// TIA Portal V15 export
// export: Created 2018-12-10T18:36:37.9324983Z, ExportSetting WithDefaults, WithReadOnly, DisplayName Totally Integrated Automation Portal, DisplayVersion V15 Update 2, DisplayName TIA Portal Openness, DisplayVersion V15 Update 2, DisplayName STEP 7 Professional, DisplayVersion V15 Update 2, DisplayName STEP 7 Safety, DisplayVersion V15, DisplayName WinCC Professional, DisplayVersion V15 Update 2, DisplayName SIMATIC Visualization Architect, DisplayVersion V15 Update 1
DATA_BLOCK "FGDB_FIXTURENAME@AddOn"   // DB132
TITLE = Geostation addon-info / Geostation Zusatz-Info
{ S7_Optimized_Access := 'FALSE' }
AUTHOR : integra
FAMILY : SYS
VERSION : 0.51
// stored: AutoNumber true, CodeModifiedDate 2017-10-24T16:57:02.4799433Z, CompileDate 2018-02-20T10:24:36.1111751Z, CreationDate 2016-12-16T08:19:31.4249609Z, DBAccessibleFromOPCUA true, InterfaceModifiedDate 2017-10-24T16:57:02.4799433Z, IsConsistent true, IsKnowHowProtected false, IsOnlyStoredInLoadMemory false, IsPLCDB false, IsWriteProtectedInAS false, ModifiedDate 2018-01-29T16:41:32.7806867Z, ParameterModified 2017-10-24T16:57:02.4799433Z, StructureModified 2017-10-24T16:57:02.4799433Z
   VAR RETAIN
      AddInfo { ExternalAccessible := 'False'; ExternalVisible := 'False'; ExternalWritable := 'False'} : Struct   // Additional informations / Zusätzliche Informationen
         "1" { ExternalAccessible := 'False'; ExternalVisible := 'False'; ExternalWritable := 'False'} : DWord;   // Additional information 1 / Zusätzliche Information 1
         "2" { ExternalAccessible := 'False'; ExternalVisible := 'False'; ExternalWritable := 'False'} : DWord;   // Additional information 2 / Zusätzliche Information 2
         "3" { ExternalAccessible := 'False'; ExternalVisible := 'False'; ExternalWritable := 'False'} : DWord;   // Additional information 3 / Zusätzliche Information 3
         "4" { ExternalAccessible := 'False'; ExternalVisible := 'False'; ExternalWritable := 'False'} : DWord;   // Additional information 4 / Zusätzliche Information 4
         "5" { ExternalAccessible := 'False'; ExternalVisible := 'False'; ExternalWritable := 'False'} : DWord;   // Additional information 5 / Zusätzliche Information 5
         "6" { ExternalAccessible := 'False'; ExternalVisible := 'False'; ExternalWritable := 'False'} : DWord;   // Additional information 6 / Zusätzliche Information 6
      END_STRUCT;
      AddT { ExternalAccessible := 'False'; ExternalVisible := 'False'; ExternalWritable := 'False'} : Struct   // Additional tags / Zusätzliche Steuervariablen
         "1" { ExternalAccessible := 'False'; ExternalVisible := 'False'; ExternalWritable := 'False'} : Bool;   // !* Additional tag 1 / !* Zusätzliche Steuervariablen 1
         "2" { ExternalAccessible := 'False'; ExternalVisible := 'False'; ExternalWritable := 'False'} : Bool;   // !* Additional tag 2 / !* Zusätzliche Steuervariablen 2
         "3" { ExternalAccessible := 'False'; ExternalVisible := 'False'; ExternalWritable := 'False'} : Bool;   // !* Additional tag 3 / !* Zusätzliche Steuervariablen 3
         "4" { ExternalAccessible := 'False'; ExternalVisible := 'False'; ExternalWritable := 'False'} : Bool;   // !* Additional tag 4 / !* Zusätzliche Steuervariablen 4
         "5" { ExternalAccessible := 'False'; ExternalVisible := 'False'; ExternalWritable := 'False'} : Bool;   // !* Additional tag 5 / !* Zusätzliche Steuervariablen 5
         "6" { ExternalAccessible := 'False'; ExternalVisible := 'False'; ExternalWritable := 'False'} : Bool;   // !* Additional tag 6 / !* Zusätzliche Steuervariablen 6
         "7" { ExternalAccessible := 'False'; ExternalVisible := 'False'; ExternalWritable := 'False'} : Bool;   // !* Additional tag 7 / !* Zusätzliche Steuervariablen 7
         "8" { ExternalAccessible := 'False'; ExternalVisible := 'False'; ExternalWritable := 'False'} : Bool;   // !* Additional tag 8 / !* Zusätzliche Steuervariablen 8
         "9" { ExternalAccessible := 'False'; ExternalVisible := 'False'; ExternalWritable := 'False'} : Bool;   // !* Additional tag 9 / !* Zusätzliche Steuervariablen 9
         "10" { ExternalAccessible := 'False'; ExternalVisible := 'False'; ExternalWritable := 'False'} : Bool;   // !* Additional tag 10 / !* Zusätzliche Steuervariablen 10
         "11" { ExternalAccessible := 'False'; ExternalVisible := 'False'; ExternalWritable := 'False'} : Bool;   // !* Additional tag 11 / !* Zusätzliche Steuervariablen 11
         "12" { ExternalAccessible := 'False'; ExternalVisible := 'False'; ExternalWritable := 'False'} : Bool;   // !* Additional tag 12 / !* Zusätzliche Steuervariablen 12
         "13" { ExternalAccessible := 'False'; ExternalVisible := 'False'; ExternalWritable := 'False'} : Bool;   // !* Additional tag 13 / !* Zusätzliche Steuervariablen 13
         "14" { ExternalAccessible := 'False'; ExternalVisible := 'False'; ExternalWritable := 'False'} : Bool;   // !* Additional tag 14 / !* Zusätzliche Steuervariablen 14
         "15" { ExternalAccessible := 'False'; ExternalVisible := 'False'; ExternalWritable := 'False'} : Bool;   // !* Additional tag 15 / !* Zusätzliche Steuervariablen 15
         "16" { ExternalAccessible := 'False'; ExternalVisible := 'False'; ExternalWritable := 'False'} : Bool;   // !* Additional tag 16 / !* Zusätzliche Steuervariablen 16
      END_STRUCT;
      AddS { ExternalAccessible := 'False'; ExternalVisible := 'False'; ExternalWritable := 'False'} : Struct   // Additional sensors / Zusätzliche Sensoren
         init_pos { ExternalAccessible := 'False'; ExternalVisible := 'False'; ExternalWritable := 'False'} : Bool;   // initial position station empty / Anfangsposition Station leer
         "2" { ExternalAccessible := 'False'; ExternalVisible := 'False'; ExternalWritable := 'False'} : Bool;   // !* Additional tag 2 / !* Zusätzliche Steuervariablen 2
         "3" { ExternalAccessible := 'False'; ExternalVisible := 'False'; ExternalWritable := 'False'} : Bool;   // !* Additional tag 3 / !* Zusätzliche Steuervariablen 3
         "4" { ExternalAccessible := 'False'; ExternalVisible := 'False'; ExternalWritable := 'False'} : Bool;   // !* Additional tag 4 / !* Zusätzliche Steuervariablen 4
         "5" { ExternalAccessible := 'False'; ExternalVisible := 'False'; ExternalWritable := 'False'} : Bool;   // !* Additional tag 5 / !* Zusätzliche Steuervariablen 5
         "6" { ExternalAccessible := 'False'; ExternalVisible := 'False'; ExternalWritable := 'False'} : Bool;   // !* Additional tag 6 / !* Zusätzliche Steuervariablen 6
         "7" { ExternalAccessible := 'False'; ExternalVisible := 'False'; ExternalWritable := 'False'} : Bool;   // !* Additional tag 7 / !* Zusätzliche Steuervariablen 7
         "8" { ExternalAccessible := 'False'; ExternalVisible := 'False'; ExternalWritable := 'False'} : Bool;   // !* Additional tag 8 / !* Zusätzliche Steuervariablen 8
         "9" { ExternalAccessible := 'False'; ExternalVisible := 'False'; ExternalWritable := 'False'} : Bool;   // !* Additional tag 9 / !* Zusätzliche Steuervariablen 9
         "10" { ExternalAccessible := 'False'; ExternalVisible := 'False'; ExternalWritable := 'False'} : Bool;   // !* Additional tag 10 / !* Zusätzliche Steuervariablen 10
         "11" { ExternalAccessible := 'False'; ExternalVisible := 'False'; ExternalWritable := 'False'} : Bool;   // !* Additional tag 11 / !* Zusätzliche Steuervariablen 11
         "12" { ExternalAccessible := 'False'; ExternalVisible := 'False'; ExternalWritable := 'False'} : Bool;   // !* Additional tag 12 / !* Zusätzliche Steuervariablen 12
         "13" { ExternalAccessible := 'False'; ExternalVisible := 'False'; ExternalWritable := 'False'} : Bool;   // !* Additional tag 13 / !* Zusätzliche Steuervariablen 13
         "14" { ExternalAccessible := 'False'; ExternalVisible := 'False'; ExternalWritable := 'False'} : Bool;   // !* Additional tag 14 / !* Zusätzliche Steuervariablen 14
         "15" { ExternalAccessible := 'False'; ExternalVisible := 'False'; ExternalWritable := 'False'} : Bool;   // !* Additional tag 15 / !* Zusätzliche Steuervariablen 15
         "16" { ExternalAccessible := 'False'; ExternalVisible := 'False'; ExternalWritable := 'False'} : Bool;   // !* Additional tag 16 / !* Zusätzliche Steuervariablen 16
      END_STRUCT;
      ExtF { ExternalAccessible := 'False'; ExternalVisible := 'False'; ExternalWritable := 'False'} : Struct   // External faults / Externe Störungen
         PartControl { ExternalAccessible := 'False'; ExternalVisible := 'False'; ExternalWritable := 'False'} : Bool;   // Part Control Error / Bauteilkontrol Fehler
         "2" { ExternalAccessible := 'False'; ExternalVisible := 'False'; ExternalWritable := 'False'} : Bool;   // !* External fault 2 / !* Externer Störung 2
         "3" { ExternalAccessible := 'False'; ExternalVisible := 'False'; ExternalWritable := 'False'} : Bool;   // !* External fault 3 / !* Externer Störung 3
         "4" { ExternalAccessible := 'False'; ExternalVisible := 'False'; ExternalWritable := 'False'} : Bool;   // !* External fault 4 / !* Externer Störung 4
         "5" { ExternalAccessible := 'False'; ExternalVisible := 'False'; ExternalWritable := 'False'} : Bool;   // !* External fault 5 / !* Externer Störung 5
         "6" { ExternalAccessible := 'False'; ExternalVisible := 'False'; ExternalWritable := 'False'} : Bool;   // !* External fault 6 / !* Externer Störung 6
         "7" { ExternalAccessible := 'False'; ExternalVisible := 'False'; ExternalWritable := 'False'} : Bool;   // !* External fault 7 / !* Externer Störung 7
         "8" { ExternalAccessible := 'False'; ExternalVisible := 'False'; ExternalWritable := 'False'} : Bool;   // !* External fault 8 / !* Externer Störung 8
         "9" { ExternalAccessible := 'False'; ExternalVisible := 'False'; ExternalWritable := 'False'} : Bool;   // !* External fault 9 / !* Externer Störung 9
         "10" { ExternalAccessible := 'False'; ExternalVisible := 'False'; ExternalWritable := 'False'} : Bool;   // !* External fault 10 / !* Externer Störung 10
         "11" { ExternalAccessible := 'False'; ExternalVisible := 'False'; ExternalWritable := 'False'} : Bool;   // !* External fault 11 / !* Externer Störung 11
         "12" { ExternalAccessible := 'False'; ExternalVisible := 'False'; ExternalWritable := 'False'} : Bool;   // !* External fault 12 / !* Externer Störung 12
         "13" { ExternalAccessible := 'False'; ExternalVisible := 'False'; ExternalWritable := 'False'} : Bool;   // !* External fault 13 / !* Externer Störung 13
         "14" { ExternalAccessible := 'False'; ExternalVisible := 'False'; ExternalWritable := 'False'} : Bool;   // !* External fault 14 / !* Externer Störung 14
         "15" { ExternalAccessible := 'False'; ExternalVisible := 'False'; ExternalWritable := 'False'} : Bool;   // !* External fault 15 / !* Externer Störung 15
         "16" { ExternalAccessible := 'False'; ExternalVisible := 'False'; ExternalWritable := 'False'} : Bool;   // !* External fault 16 / !* Externer Störung 16
      END_STRUCT;
      TransExtF { ExternalAccessible := 'False'; ExternalVisible := 'False'; ExternalWritable := 'False'} : Struct   // Transfer external faults / Übergabe externe Störungen
         PartControl { ExternalAccessible := 'False'; ExternalVisible := 'False'; ExternalWritable := 'False'} : Bool;   // Transfer external fault PartControl / Übergabe externer Störung Bauteilkontrol
         "2" { ExternalAccessible := 'False'; ExternalVisible := 'False'; ExternalWritable := 'False'} : Bool;   // Transfer external fault 2 / Übergabe externer Störung 2
         "3" { ExternalAccessible := 'False'; ExternalVisible := 'False'; ExternalWritable := 'False'} : Bool;   // Transfer external fault 3 / Übergabe externer Störung 3
         "4" { ExternalAccessible := 'False'; ExternalVisible := 'False'; ExternalWritable := 'False'} : Bool;   // Transfer external fault 4 / Übergabe externer Störung 4
         "5" { ExternalAccessible := 'False'; ExternalVisible := 'False'; ExternalWritable := 'False'} : Bool;   // Transfer external fault 5 / Übergabe externer Störung 5
         "6" { ExternalAccessible := 'False'; ExternalVisible := 'False'; ExternalWritable := 'False'} : Bool;   // Transfer external fault 6 / Übergabe externer Störung 6
         "7" { ExternalAccessible := 'False'; ExternalVisible := 'False'; ExternalWritable := 'False'} : Bool;   // Transfer external fault 7 / Übergabe externer Störung 7
         "8" { ExternalAccessible := 'False'; ExternalVisible := 'False'; ExternalWritable := 'False'} : Bool;   // Transfer external fault 8 / Übergabe externer Störung 8
         "9" { ExternalAccessible := 'False'; ExternalVisible := 'False'; ExternalWritable := 'False'} : Bool;   // Transfer external fault 9 / Übergabe externer Störung 9
         "10" { ExternalAccessible := 'False'; ExternalVisible := 'False'; ExternalWritable := 'False'} : Bool;   // Transfer external fault 10 / Übergabe externer Störung 10
         "11" { ExternalAccessible := 'False'; ExternalVisible := 'False'; ExternalWritable := 'False'} : Bool;   // Transfer external fault 11 / Übergabe externer Störung 11
         "12" { ExternalAccessible := 'False'; ExternalVisible := 'False'; ExternalWritable := 'False'} : Bool;   // Transfer external fault 12 / Übergabe externer Störung 12
         "13" { ExternalAccessible := 'False'; ExternalVisible := 'False'; ExternalWritable := 'False'} : Bool;   // Transfer external fault 13 / Übergabe externer Störung 13
         "14" { ExternalAccessible := 'False'; ExternalVisible := 'False'; ExternalWritable := 'False'} : Bool;   // Transfer external fault 14 / Übergabe externer Störung 14
         "15" { ExternalAccessible := 'False'; ExternalVisible := 'False'; ExternalWritable := 'False'} : Bool;   // Transfer external fault 15 / Übergabe externer Störung 15
         "16" { ExternalAccessible := 'False'; ExternalVisible := 'False'; ExternalWritable := 'False'} : Bool;   // Transfer external fault 16 / Übergabe externer Störung 16
      END_STRUCT;
      ExtW { ExternalAccessible := 'False'; ExternalVisible := 'False'; ExternalWritable := 'False'} : Struct   // External warnings / Externe Warnungen
         "1" { ExternalAccessible := 'False'; ExternalVisible := 'False'; ExternalWritable := 'False'} : Bool;   // !* External warning 1 / !* Externe Warnung 1
         "2" { ExternalAccessible := 'False'; ExternalVisible := 'False'; ExternalWritable := 'False'} : Bool;   // !* External warning 2 / !* Externe Warnung 2
         "3" { ExternalAccessible := 'False'; ExternalVisible := 'False'; ExternalWritable := 'False'} : Bool;   // !* External warning 3 / !* Externe Warnung 3
         "4" { ExternalAccessible := 'False'; ExternalVisible := 'False'; ExternalWritable := 'False'} : Bool;   // !* External warning 4 / !* Externe Warnung 4
         "5" { ExternalAccessible := 'False'; ExternalVisible := 'False'; ExternalWritable := 'False'} : Bool;   // !* External warning 5 / !* Externe Warnung 5
         "6" { ExternalAccessible := 'False'; ExternalVisible := 'False'; ExternalWritable := 'False'} : Bool;   // !* External warning 6 / !* Externe Warnung 6
         "7" { ExternalAccessible := 'False'; ExternalVisible := 'False'; ExternalWritable := 'False'} : Bool;   // !* External warning 7 / !* Externe Warnung 7
         "8" { ExternalAccessible := 'False'; ExternalVisible := 'False'; ExternalWritable := 'False'} : Bool;   // !* External warning 7 / !* Externe Warnung 7
      END_STRUCT;
      TransExtW { ExternalAccessible := 'False'; ExternalVisible := 'False'; ExternalWritable := 'False'} : Struct   // Transfer external warnings / Übergabe externe Warnungen
         "1" { ExternalAccessible := 'False'; ExternalVisible := 'False'; ExternalWritable := 'False'} : Bool;   // Transfer external warning 1 / Übergabe externe Warnung 1
         "2" { ExternalAccessible := 'False'; ExternalVisible := 'False'; ExternalWritable := 'False'} : Bool;   // Transfer external warning 2 / Übergabe externe Warnung 2
         "3" { ExternalAccessible := 'False'; ExternalVisible := 'False'; ExternalWritable := 'False'} : Bool;   // Transfer external warning 3 / Übergabe externe Warnung 3
         "4" { ExternalAccessible := 'False'; ExternalVisible := 'False'; ExternalWritable := 'False'} : Bool;   // Transfer external warning 4 / Übergabe externe Warnung 4
         "5" { ExternalAccessible := 'False'; ExternalVisible := 'False'; ExternalWritable := 'False'} : Bool;   // Transfer external warning 5 / Übergabe externe Warnung 5
         "6" { ExternalAccessible := 'False'; ExternalVisible := 'False'; ExternalWritable := 'False'} : Bool;   // Transfer external warning 6 / Übergabe externe Warnung 6
         "7" { ExternalAccessible := 'False'; ExternalVisible := 'False'; ExternalWritable := 'False'} : Bool;   // Transfer external warning 7 / Übergabe externe Warnung 7
         "8" { ExternalAccessible := 'False'; ExternalVisible := 'False'; ExternalWritable := 'False'} : Bool;   // Transfer external warning 8 / Übergabe externe Warnung 8
      END_STRUCT;
      ExtM { ExternalAccessible := 'False'; ExternalVisible := 'False'; ExternalWritable := 'False'} : Struct   // External messages / Externe Meldungen
         "1" { ExternalAccessible := 'False'; ExternalVisible := 'False'; ExternalWritable := 'False'} : Bool;   // !* External message 1 / !* Externe Meldung 1
         "2" { ExternalAccessible := 'False'; ExternalVisible := 'False'; ExternalWritable := 'False'} : Bool;   // !* External message 2 / !* Externe Meldung 2
         "3" { ExternalAccessible := 'False'; ExternalVisible := 'False'; ExternalWritable := 'False'} : Bool;   // !* External message 3 / !* Externe Meldung 3
         "4" { ExternalAccessible := 'False'; ExternalVisible := 'False'; ExternalWritable := 'False'} : Bool;   // !* External message 4 / !* Externe Meldung 4
         "5" { ExternalAccessible := 'False'; ExternalVisible := 'False'; ExternalWritable := 'False'} : Bool;   // !* External message 5 / !* Externe Meldung 5
         "6" { ExternalAccessible := 'False'; ExternalVisible := 'False'; ExternalWritable := 'False'} : Bool;   // !* External message 6 / !* Externe Meldung 6
         "7" { ExternalAccessible := 'False'; ExternalVisible := 'False'; ExternalWritable := 'False'} : Bool;   // !* External message 7 / !* Externe Meldung 7
         "8" { ExternalAccessible := 'False'; ExternalVisible := 'False'; ExternalWritable := 'False'} : Bool;   // !* External message 8 / !* Externe Meldung 8
      END_STRUCT;
      TransExtM { ExternalAccessible := 'False'; ExternalVisible := 'False'; ExternalWritable := 'False'} : Struct   // Transfer external messages / Übergabe externe Meldungen
         "1" { ExternalAccessible := 'False'; ExternalVisible := 'False'; ExternalWritable := 'False'} : Bool;   // Transfer external message 1 / Übergabe externe Meldung 1
         "2" { ExternalAccessible := 'False'; ExternalVisible := 'False'; ExternalWritable := 'False'} : Bool;   // Transfer external message 2 / Übergabe externe Meldung 2
         "3" { ExternalAccessible := 'False'; ExternalVisible := 'False'; ExternalWritable := 'False'} : Bool;   // Transfer external message 3 / Übergabe externe Meldung 3
         "4" { ExternalAccessible := 'False'; ExternalVisible := 'False'; ExternalWritable := 'False'} : Bool;   // Transfer external message 4 / Übergabe externe Meldung 4
         "5" { ExternalAccessible := 'False'; ExternalVisible := 'False'; ExternalWritable := 'False'} : Bool;   // Transfer external message 5 / Übergabe externe Meldung 5
         "6" { ExternalAccessible := 'False'; ExternalVisible := 'False'; ExternalWritable := 'False'} : Bool;   // Transfer external message 6 / Übergabe externe Meldung 6
         "7" { ExternalAccessible := 'False'; ExternalVisible := 'False'; ExternalWritable := 'False'} : Bool;   // Transfer external message 7 / Übergabe externe Meldung 7
         "8" { ExternalAccessible := 'False'; ExternalVisible := 'False'; ExternalWritable := 'False'} : Bool;   // Transfer external message 8 / Übergabe externe Meldung 8
      END_STRUCT;
      ES { ExternalAccessible := 'False'; ExternalVisible := 'False'; ExternalWritable := 'False'} : Struct   // Emergeny stops / Not-Halt
         "1" { ExternalAccessible := 'False'; ExternalVisible := 'False'; ExternalWritable := 'False'} : Bool;   // !* Emergency stop 1 / !* Not-Halt 1
         "2" { ExternalAccessible := 'False'; ExternalVisible := 'False'; ExternalWritable := 'False'} : Bool;   // !* Emergency stop 2 / !* Not-Halt 2
         "3" { ExternalAccessible := 'False'; ExternalVisible := 'False'; ExternalWritable := 'False'} : Bool;   // !* Emergency stop 3 / !* Not-Halt 3
         "4" { ExternalAccessible := 'False'; ExternalVisible := 'False'; ExternalWritable := 'False'} : Bool;   // !* Emergency stop 4 / !* Not-Halt 4
         "5" { ExternalAccessible := 'False'; ExternalVisible := 'False'; ExternalWritable := 'False'} : Bool;   // !* Emergency stop 5 / !* Not-Halt 5
         "6" { ExternalAccessible := 'False'; ExternalVisible := 'False'; ExternalWritable := 'False'} : Bool;   // !* Emergency stop 6 / !* Not-Halt 6
         "7" { ExternalAccessible := 'False'; ExternalVisible := 'False'; ExternalWritable := 'False'} : Bool;   // !* Emergency stop 7 / !* Not-Halt 7
         "8" { ExternalAccessible := 'False'; ExternalVisible := 'False'; ExternalWritable := 'False'} : Bool;   // !* Emergency stop 8 / !* Not-Halt 8
      END_STRUCT;
      TransES { ExternalAccessible := 'False'; ExternalVisible := 'False'; ExternalWritable := 'False'} : Struct   // Transfer Emergeny stops / Übergabe Not-Halt
         "1" { ExternalAccessible := 'False'; ExternalVisible := 'False'; ExternalWritable := 'False'} : Bool;   // Transfer Emergeny stop 1 / Übergabe Not-Halt 1
         "2" { ExternalAccessible := 'False'; ExternalVisible := 'False'; ExternalWritable := 'False'} : Bool;   // Transfer Emergeny stop 2 / Übergabe Not-Halt 2
         "3" { ExternalAccessible := 'False'; ExternalVisible := 'False'; ExternalWritable := 'False'} : Bool;   // Transfer Emergeny stop 3 / Übergabe Not-Halt 3
         "4" { ExternalAccessible := 'False'; ExternalVisible := 'False'; ExternalWritable := 'False'} : Bool;   // Transfer Emergeny stop 4 / Übergabe Not-Halt 4
         "5" { ExternalAccessible := 'False'; ExternalVisible := 'False'; ExternalWritable := 'False'} : Bool;   // Transfer Emergeny stop 5 / Übergabe Not-Halt 5
         "6" { ExternalAccessible := 'False'; ExternalVisible := 'False'; ExternalWritable := 'False'} : Bool;   // Transfer Emergeny stop 6 / Übergabe Not-Halt 6
         "7" { ExternalAccessible := 'False'; ExternalVisible := 'False'; ExternalWritable := 'False'} : Bool;   // Transfer Emergeny stop 7 / Übergabe Not-Halt 7
         "8" { ExternalAccessible := 'False'; ExternalVisible := 'False'; ExternalWritable := 'False'} : Bool;   // Transfer Emergeny stop 8 / Übergabe Not-Halt 8
      END_STRUCT;
      Masks { ExternalAccessible := 'False'; ExternalVisible := 'False'; ExternalWritable := 'False'} : Struct   // Masks / Masken
         prodRelevantFault1_8 { ExternalAccessible := 'False'; ExternalVisible := 'False'; ExternalWritable := 'False'} : Byte;   // * Mask external fault 1-8 (0=production-rel.) / * Maske externe Störungen 1- 8 (0=produktionsrel.)
         prodRelevantFault9_16 { ExternalAccessible := 'False'; ExternalVisible := 'False'; ExternalWritable := 'False'} : Byte;   // * Mask external fault 9-16 (0=production-rel.) / * Maske externe Störungen 9- 16 (0=produktionsrel.)
         prodRelevantWarning1_8 { ExternalAccessible := 'False'; ExternalVisible := 'False'; ExternalWritable := 'False'} : Byte;   // * Mask external warning 1-8 (0=production-rel.) / * Maske externe Warnungen 1- 8 (0=produktionsrel.)
         prodRelevantMessage1_8 { ExternalAccessible := 'False'; ExternalVisible := 'False'; ExternalWritable := 'False'} : Byte;   // * Mask external message 1-8 (0=production-rel.) / * Maske externe Meldungen 1- 8 (0=produktionsrel.)
      END_STRUCT;
      GroupMessages { ExternalAccessible := 'False'; ExternalVisible := 'False'; ExternalWritable := 'False'} : Struct   // Group messages / Sammelmeldungen
         groupMessageFault1_8 { ExternalAccessible := 'False'; ExternalVisible := 'False'; ExternalWritable := 'False'} : Bool;   // Group message external fault 1-8 / Sammelmeldung externe Störung 1-8
         groupMessageFault9_16 { ExternalAccessible := 'False'; ExternalVisible := 'False'; ExternalWritable := 'False'} : Bool;   // Group message external fault 9-16 / Sammelmeldung externe Störung 9-16
         groupMessageWarning1_8 { ExternalAccessible := 'False'; ExternalVisible := 'False'; ExternalWritable := 'False'} : Bool;   // Group message external warning 1-8 / Sammelmeldung externe Warnung 1-8
         groupMessageMessage1_8 { ExternalAccessible := 'False'; ExternalVisible := 'False'; ExternalWritable := 'False'} : Bool;   // Group message external message 1-8 / Sammelmeldung externe Meldung 1-8
      END_STRUCT;
   END_VAR
BEGIN
END_DATA_BLOCK
